// TIA Portal project "SepSimples" (V16)

(* hardware
DEVICE "S71500/ET200MP station_1"  S7-1500 station
   slot 0: "Rail_0"  Rack  6ES7 590-1***0-0AA0
   slot 1: "PLC_1"  CPU 1512C-1 PN  6ES7 512-1CK00-0AB0  V2.8
      slot 3: "CPU display_1"  6ES7591-1AA00-0AA0
      slot 32768: "PROFINET interface_1"  X1
         slot 32769: "Port_1"  X1 P1
         slot 32770: "Port_2"  X1 P2
      slot 34817: "Virtual CP interface port_1"  Virtual CP interface port  Virtual CP interface port
*)

// ===== PLC "PLC_1"  CPU 1512C-1 PN =====

VAR_GLOBAL   // PLC tag table "Default tag table"
   "alwaysFalse" AT %M0.0 : Bool;
END_VAR

VAR_GLOBAL   // PLC tag table "E_N_Controlavel"
   "FIO_S3" AT %M5.3 : Bool;
   "FIO_S2" AT %M5.2 : Bool;
   "FIO_PA" AT %M5.1 : Bool;
   "FIO_PV" AT %M5.0 : Bool;
   "FIO_S4" AT %M5.5 : Bool;
   "FIO_AT_Fwd" AT %M5.6 : Bool;
   "FIOAT_Rev" AT %M5.7 : Bool;
END_VAR

VAR_GLOBAL   // PLC tag table "Saidas"
   "FIO_Atuador" AT %M10.0 : Bool;
   "FIO_Esteira1" AT %M10.1 : Bool;
   "FIO_Esteira2" AT %M10.2 : Bool;
   "FIO_Esteira3" AT %M10.3 : Bool;
   "FIO_Esteira4" AT %M10.4 : Bool;
END_VAR

DATA_BLOCK "Eventos"   // DB1
{ S7_Optimized_Access := 'TRUE' }
VERSION : 0.1
   VAR
      PV_Ev : Bool;
      PA_Ev : Bool;
      S2_On_Ev : Bool;
      S2_Off_Ev : Bool;
      S3_On_Ev : Bool;
      S3_Off_Ev : Bool;
      AT_Off_Ev : Bool;
      S4_Off_Ev : Bool;
      AT_On_Ev : Bool;
      E1_On_Ev : Bool;
      E1_Off_Ev : Bool;
      E2_On_Ev : Bool;
      E2_Off_Ev : Bool;
      E3_On_Ev : Bool;
      E3_Off_Ev : Bool;
   END_VAR
BEGIN
END_DATA_BLOCK

DATA_BLOCK "BitsAuxiliares"   // DB2
{ S7_Optimized_Access := 'TRUE' }
VERSION : 0.1
   VAR
      Aux1 : Bool;
      Aux2 : Bool;
      Aux3 : Bool;
      Aux4 : Bool;
      Aux5 : Bool;
      Aux6 : Bool;
      Aux7 : Bool;
      Aux8 : Bool;
   END_VAR
BEGIN
END_DATA_BLOCK

DATA_BLOCK "EstadosSP"   // DB3
{ S7_Optimized_Access := 'TRUE' }
VERSION : 0.1
   VAR
      GS1_1 : Bool := true;
      GS2_1 : Bool := true;
      GS2_2 : Bool;
      GS3_1 : Bool := true;
      GS3_2 : Bool;
      GAT_1 : Bool := true;
      GAT_2 : Bool;
      GE1_1 : Bool := true;
      GE1_2 : Bool;
      GE2_1 : Bool := true;
      GE2_2 : Bool;
      GE3_1 : Bool := true;
      GE3_2 : Bool;
      GS4_1 : Bool := true;
   END_VAR
BEGIN
END_DATA_BLOCK

DATA_BLOCK "EstadosSup"   // DB4
{ S7_Optimized_Access := 'TRUE' }
VERSION : 0.1
   VAR
      Sup1_1 : Bool := true;
      Sup1_2 : Bool;
      Sup2_1 : Bool := true;
      Sup2_2 : Bool;
      Sup3_1 : Bool := true;
      Sup3_2 : Bool;
      Sup4_1 : Bool := true;
      Sup4_2 : Bool;
      Sup5_1 : Bool := true;
      Sup5_2 : Bool;
      Sup6_1 : Bool := true;
      Sup6_2 : Bool;
      Sup7_1 : Bool := true;
      Sup7_2 : Bool;
      Sup8_1 : Bool := true;
      Sup8_2 : Bool;
      Sup9_1 : Bool := true;
      Sup9_2 : Bool;
      Sup9_3 : Bool;
      Sup10_1 : Bool := true;
      Sup10_2 : Bool;
      Sup10_3 : Bool;
      Sup10_4 : Bool;
   END_VAR
BEGIN
END_DATA_BLOCK

DATA_BLOCK "Des_Eventos"   // DB5
{ S7_Optimized_Access := 'TRUE' }
VERSION : 0.1
   VAR
      d_AT_On : Bool;
      d_E1_On : Bool;
      d_E1_Off : Bool;
      d_E2_On : Bool;
      d_E2_Off : Bool;
      d_E3_On : Bool;
      d_E3_Off : Bool;
   END_VAR
BEGIN
END_DATA_BLOCK

FUNCTION "LeituraEntradas" : Void   // FC2, LAD
TITLE = Leitura das entradas dos eventos não controláveis
{ S7_Optimized_Access := 'TRUE' }
VERSION : 0.1
   VAR_TEMP   // added for the SCL form of the ladder/FBD networks
      _w1 : Bool;
   END_VAR
BEGIN

REGION Network 1: Leitura peça verde
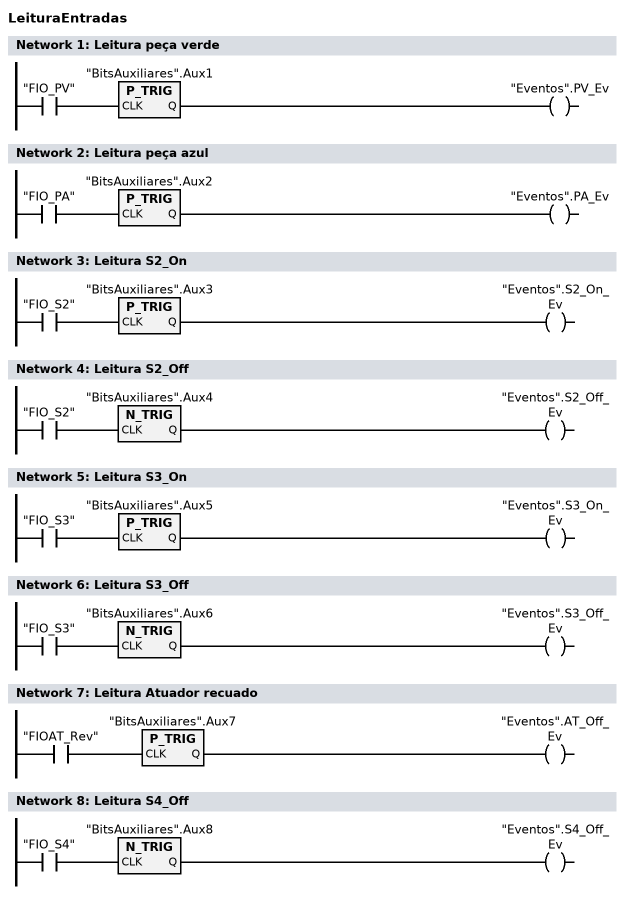
   RUNG wire#powerrail
      Contact( "FIO_PV" )
      P_Trig( "BitsAuxiliares".Aux1 )
      Coil( "Eventos".PV_Ev )
   END_RUNG
   // the same network as SCL:
   #_w1 := "FIO_PV" AND NOT "BitsAuxiliares".Aux1;   // rising edge
   "BitsAuxiliares".Aux1 := "FIO_PV";
   "Eventos".PV_Ev := #_w1;
END_REGION

REGION Network 2: Leitura peça azul
   RUNG wire#powerrail
      Contact( "FIO_PA" )
      P_Trig( "BitsAuxiliares".Aux2 )
      Coil( "Eventos".PA_Ev )
   END_RUNG
   // the same network as SCL:
   #_w1 := "FIO_PA" AND NOT "BitsAuxiliares".Aux2;   // rising edge
   "BitsAuxiliares".Aux2 := "FIO_PA";
   "Eventos".PA_Ev := #_w1;
END_REGION

REGION Network 3: Leitura S2_On
   RUNG wire#powerrail
      Contact( "FIO_S2" )
      P_Trig( "BitsAuxiliares".Aux3 )
      Coil( "Eventos".S2_On_Ev )
   END_RUNG
   // the same network as SCL:
   #_w1 := "FIO_S2" AND NOT "BitsAuxiliares".Aux3;   // rising edge
   "BitsAuxiliares".Aux3 := "FIO_S2";
   "Eventos".S2_On_Ev := #_w1;
END_REGION

REGION Network 4: Leitura S2_Off
   RUNG wire#powerrail
      Contact( "FIO_S2" )
      N_Trig( "BitsAuxiliares".Aux4 )
      Coil( "Eventos".S2_Off_Ev )
   END_RUNG
   // the same network as SCL:
   #_w1 := NOT "FIO_S2" AND "BitsAuxiliares".Aux4;   // falling edge
   "BitsAuxiliares".Aux4 := "FIO_S2";
   "Eventos".S2_Off_Ev := #_w1;
END_REGION

REGION Network 5: Leitura S3_On
   RUNG wire#powerrail
      Contact( "FIO_S3" )
      P_Trig( "BitsAuxiliares".Aux5 )
      Coil( "Eventos".S3_On_Ev )
   END_RUNG
   // the same network as SCL:
   #_w1 := "FIO_S3" AND NOT "BitsAuxiliares".Aux5;   // rising edge
   "BitsAuxiliares".Aux5 := "FIO_S3";
   "Eventos".S3_On_Ev := #_w1;
END_REGION

REGION Network 6: Leitura S3_Off
   RUNG wire#powerrail
      Contact( "FIO_S3" )
      N_Trig( "BitsAuxiliares".Aux6 )
      Coil( "Eventos".S3_Off_Ev )
   END_RUNG
   // the same network as SCL:
   #_w1 := NOT "FIO_S3" AND "BitsAuxiliares".Aux6;   // falling edge
   "BitsAuxiliares".Aux6 := "FIO_S3";
   "Eventos".S3_Off_Ev := #_w1;
END_REGION

REGION Network 7: Leitura Atuador recuado
   RUNG wire#powerrail
      Contact( "FIOAT_Rev" )
      P_Trig( "BitsAuxiliares".Aux7 )
      Coil( "Eventos".AT_Off_Ev )
   END_RUNG
   // the same network as SCL:
   #_w1 := "FIOAT_Rev" AND NOT "BitsAuxiliares".Aux7;   // rising edge
   "BitsAuxiliares".Aux7 := "FIOAT_Rev";
   "Eventos".AT_Off_Ev := #_w1;
END_REGION

REGION Network 8: Leitura S4_Off
   RUNG wire#powerrail
      Contact( "FIO_S4" )
      N_Trig( "BitsAuxiliares".Aux8 )
      Coil( "Eventos".S4_Off_Ev )
   END_RUNG
   // the same network as SCL:
   #_w1 := NOT "FIO_S4" AND "BitsAuxiliares".Aux8;   // falling edge
   "BitsAuxiliares".Aux8 := "FIO_S4";
   "Eventos".S4_Off_Ev := #_w1;
END_REGION
END_FUNCTION

FUNCTION "At_SP_NaoControlaveis" : Void   // FC3, LAD
TITLE = Atualização dos estados do sistema produto a partir dos eventos não controláveis.
{ S7_Optimized_Access := 'TRUE' }
VERSION : 0.1
BEGIN

REGION Network 1: Modelo de S2, do estado 1 para o estado 2.
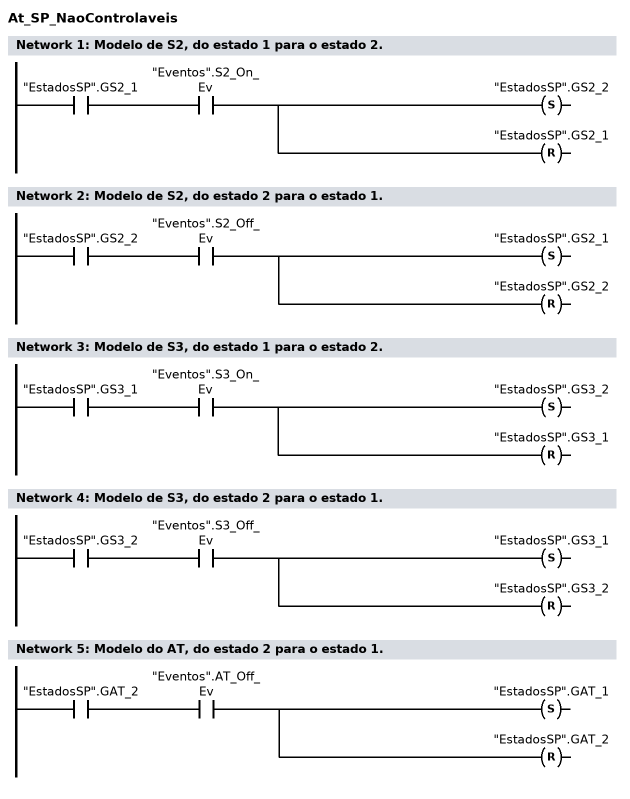
   RUNG wire#powerrail
      Contact( "EstadosSP".GS2_1 )
      Contact( "Eventos".S2_On_Ev )
      wire#w1
      S_Coil( "EstadosSP".GS2_2 )
   END_RUNG
   RUNG wire#w1
      R_Coil( "EstadosSP".GS2_1 )
   END_RUNG
   // the same network as SCL:
   IF "EstadosSP".GS2_1 AND "Eventos".S2_On_Ev THEN
       "EstadosSP".GS2_2 := TRUE;
       "EstadosSP".GS2_1 := FALSE;
   END_IF;
END_REGION

REGION Network 2: Modelo de S2, do estado 2 para o estado 1.
   RUNG wire#powerrail
      Contact( "EstadosSP".GS2_2 )
      Contact( "Eventos".S2_Off_Ev )
      wire#w1
      S_Coil( "EstadosSP".GS2_1 )
   END_RUNG
   RUNG wire#w1
      R_Coil( "EstadosSP".GS2_2 )
   END_RUNG
   // the same network as SCL:
   IF "EstadosSP".GS2_2 AND "Eventos".S2_Off_Ev THEN
       "EstadosSP".GS2_1 := TRUE;
       "EstadosSP".GS2_2 := FALSE;
   END_IF;
END_REGION

REGION Network 3: Modelo de S3, do estado 1 para o estado 2.
   RUNG wire#powerrail
      Contact( "EstadosSP".GS3_1 )
      Contact( "Eventos".S3_On_Ev )
      wire#w1
      S_Coil( "EstadosSP".GS3_2 )
   END_RUNG
   RUNG wire#w1
      R_Coil( "EstadosSP".GS3_1 )
   END_RUNG
   // the same network as SCL:
   IF "EstadosSP".GS3_1 AND "Eventos".S3_On_Ev THEN
       "EstadosSP".GS3_2 := TRUE;
       "EstadosSP".GS3_1 := FALSE;
   END_IF;
END_REGION

REGION Network 4: Modelo de S3, do estado 2 para o estado 1.
   RUNG wire#powerrail
      Contact( "EstadosSP".GS3_2 )
      Contact( "Eventos".S3_Off_Ev )
      wire#w1
      S_Coil( "EstadosSP".GS3_1 )
   END_RUNG
   RUNG wire#w1
      R_Coil( "EstadosSP".GS3_2 )
   END_RUNG
   // the same network as SCL:
   IF "EstadosSP".GS3_2 AND "Eventos".S3_Off_Ev THEN
       "EstadosSP".GS3_1 := TRUE;
       "EstadosSP".GS3_2 := FALSE;
   END_IF;
END_REGION

REGION Network 5: Modelo do AT, do estado 2 para o estado 1.
   RUNG wire#powerrail
      Contact( "EstadosSP".GAT_2 )
      Contact( "Eventos".AT_Off_Ev )
      wire#w1
      S_Coil( "EstadosSP".GAT_1 )
   END_RUNG
   RUNG wire#w1
      R_Coil( "EstadosSP".GAT_2 )
   END_RUNG
   // the same network as SCL:
   IF "EstadosSP".GAT_2 AND "Eventos".AT_Off_Ev THEN
       "EstadosSP".GAT_1 := TRUE;
       "EstadosSP".GAT_2 := FALSE;
   END_IF;
END_REGION
END_FUNCTION

FUNCTION "At_Sup_NaoControlaveis" : Void   // FC4, LAD
TITLE = Atualização dos estados dos supervisores reduzidos, devido a eventos não controláveis
{ S7_Optimized_Access := 'TRUE' }
VERSION : 0.1
BEGIN

REGION Network 1: Atualização do supervisor 1, estado 2 para estado 1.
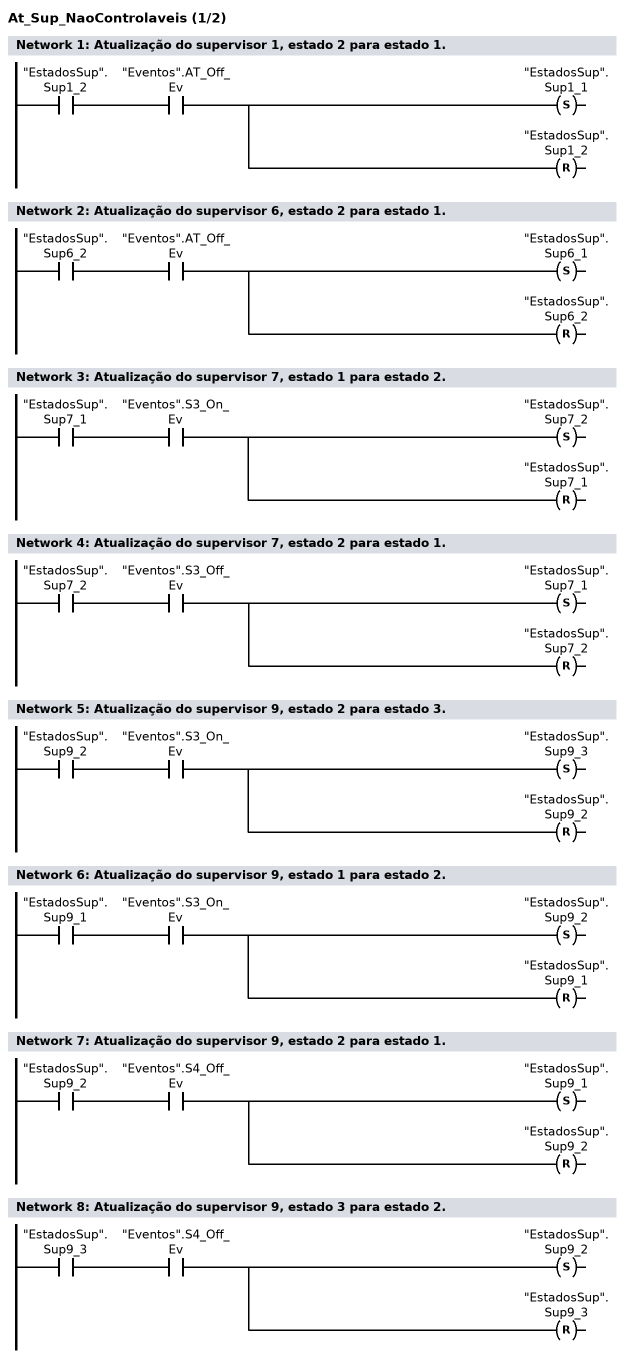
   RUNG wire#powerrail
      Contact( "EstadosSup".Sup1_2 )
      Contact( "Eventos".AT_Off_Ev )
      wire#w1
      S_Coil( "EstadosSup".Sup1_1 )
   END_RUNG
   RUNG wire#w1
      R_Coil( "EstadosSup".Sup1_2 )
   END_RUNG
   // the same network as SCL:
   IF "EstadosSup".Sup1_2 AND "Eventos".AT_Off_Ev THEN
       "EstadosSup".Sup1_1 := TRUE;
       "EstadosSup".Sup1_2 := FALSE;
   END_IF;
END_REGION

REGION Network 2: Atualização do supervisor 6, estado 2 para estado 1.
   RUNG wire#powerrail
      Contact( "EstadosSup".Sup6_2 )
      Contact( "Eventos".AT_Off_Ev )
      wire#w1
      S_Coil( "EstadosSup".Sup6_1 )
   END_RUNG
   RUNG wire#w1
      R_Coil( "EstadosSup".Sup6_2 )
   END_RUNG
   // the same network as SCL:
   IF "EstadosSup".Sup6_2 AND "Eventos".AT_Off_Ev THEN
       "EstadosSup".Sup6_1 := TRUE;
       "EstadosSup".Sup6_2 := FALSE;
   END_IF;
END_REGION

REGION Network 3: Atualização do supervisor 7, estado 1 para estado 2.
   RUNG wire#powerrail
      Contact( "EstadosSup".Sup7_1 )
      Contact( "Eventos".S3_On_Ev )
      wire#w1
      S_Coil( "EstadosSup".Sup7_2 )
   END_RUNG
   RUNG wire#w1
      R_Coil( "EstadosSup".Sup7_1 )
   END_RUNG
   // the same network as SCL:
   IF "EstadosSup".Sup7_1 AND "Eventos".S3_On_Ev THEN
       "EstadosSup".Sup7_2 := TRUE;
       "EstadosSup".Sup7_1 := FALSE;
   END_IF;
END_REGION

REGION Network 4: Atualização do supervisor 7, estado 2 para estado 1.
   RUNG wire#powerrail
      Contact( "EstadosSup".Sup7_2 )
      Contact( "Eventos".S3_Off_Ev )
      wire#w1
      S_Coil( "EstadosSup".Sup7_1 )
   END_RUNG
   RUNG wire#w1
      R_Coil( "EstadosSup".Sup7_2 )
   END_RUNG
   // the same network as SCL:
   IF "EstadosSup".Sup7_2 AND "Eventos".S3_Off_Ev THEN
       "EstadosSup".Sup7_1 := TRUE;
       "EstadosSup".Sup7_2 := FALSE;
   END_IF;
END_REGION

REGION Network 5: Atualização do supervisor 9, estado 2 para estado 3.
   RUNG wire#powerrail
      Contact( "EstadosSup".Sup9_2 )
      Contact( "Eventos".S3_On_Ev )
      wire#w1
      S_Coil( "EstadosSup".Sup9_3 )
   END_RUNG
   RUNG wire#w1
      R_Coil( "EstadosSup".Sup9_2 )
   END_RUNG
   // the same network as SCL:
   IF "EstadosSup".Sup9_2 AND "Eventos".S3_On_Ev THEN
       "EstadosSup".Sup9_3 := TRUE;
       "EstadosSup".Sup9_2 := FALSE;
   END_IF;
END_REGION

REGION Network 6: Atualização do supervisor 9, estado 1 para estado 2.
   RUNG wire#powerrail
      Contact( "EstadosSup".Sup9_1 )
      Contact( "Eventos".S3_On_Ev )
      wire#w1
      S_Coil( "EstadosSup".Sup9_2 )
   END_RUNG
   RUNG wire#w1
      R_Coil( "EstadosSup".Sup9_1 )
   END_RUNG
   // the same network as SCL:
   IF "EstadosSup".Sup9_1 AND "Eventos".S3_On_Ev THEN
       "EstadosSup".Sup9_2 := TRUE;
       "EstadosSup".Sup9_1 := FALSE;
   END_IF;
END_REGION

REGION Network 7: Atualização do supervisor 9, estado 2 para estado 1.
   RUNG wire#powerrail
      Contact( "EstadosSup".Sup9_2 )
      Contact( "Eventos".S4_Off_Ev )
      wire#w1
      S_Coil( "EstadosSup".Sup9_1 )
   END_RUNG
   RUNG wire#w1
      R_Coil( "EstadosSup".Sup9_2 )
   END_RUNG
   // the same network as SCL:
   IF "EstadosSup".Sup9_2 AND "Eventos".S4_Off_Ev THEN
       "EstadosSup".Sup9_1 := TRUE;
       "EstadosSup".Sup9_2 := FALSE;
   END_IF;
END_REGION

REGION Network 8: Atualização do supervisor 9, estado 3 para estado 2.
   RUNG wire#powerrail
      Contact( "EstadosSup".Sup9_3 )
      Contact( "Eventos".S4_Off_Ev )
      wire#w1
      S_Coil( "EstadosSup".Sup9_2 )
   END_RUNG
   RUNG wire#w1
      R_Coil( "EstadosSup".Sup9_3 )
   END_RUNG
   // the same network as SCL:
   IF "EstadosSup".Sup9_3 AND "Eventos".S4_Off_Ev THEN
       "EstadosSup".Sup9_2 := TRUE;
       "EstadosSup".Sup9_3 := FALSE;
   END_IF;
END_REGION

REGION Network 9: Atualização do supervisor 10, estado 1 para estado 2.
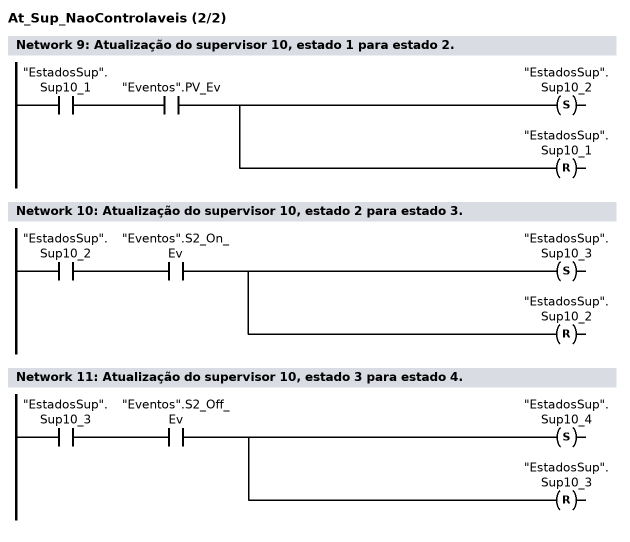
   RUNG wire#powerrail
      Contact( "EstadosSup".Sup10_1 )
      Contact( "Eventos".PV_Ev )
      wire#w1
      S_Coil( "EstadosSup".Sup10_2 )
   END_RUNG
   RUNG wire#w1
      R_Coil( "EstadosSup".Sup10_1 )
   END_RUNG
   // the same network as SCL:
   IF "EstadosSup".Sup10_1 AND "Eventos".PV_Ev THEN
       "EstadosSup".Sup10_2 := TRUE;
       "EstadosSup".Sup10_1 := FALSE;
   END_IF;
END_REGION

REGION Network 10: Atualização do supervisor 10, estado 2 para estado 3.
   RUNG wire#powerrail
      Contact( "EstadosSup".Sup10_2 )
      Contact( "Eventos".S2_On_Ev )
      wire#w1
      S_Coil( "EstadosSup".Sup10_3 )
   END_RUNG
   RUNG wire#w1
      R_Coil( "EstadosSup".Sup10_2 )
   END_RUNG
   // the same network as SCL:
   IF "EstadosSup".Sup10_2 AND "Eventos".S2_On_Ev THEN
       "EstadosSup".Sup10_3 := TRUE;
       "EstadosSup".Sup10_2 := FALSE;
   END_IF;
END_REGION

REGION Network 11: Atualização do supervisor 10, estado 3 para estado 4.
   RUNG wire#powerrail
      Contact( "EstadosSup".Sup10_3 )
      Contact( "Eventos".S2_Off_Ev )
      wire#w1
      S_Coil( "EstadosSup".Sup10_4 )
   END_RUNG
   RUNG wire#w1
      R_Coil( "EstadosSup".Sup10_3 )
   END_RUNG
   // the same network as SCL:
   IF "EstadosSup".Sup10_3 AND "Eventos".S2_Off_Ev THEN
       "EstadosSup".Sup10_4 := TRUE;
       "EstadosSup".Sup10_3 := FALSE;
   END_IF;
END_REGION
END_FUNCTION

FUNCTION "Des_EventosControlaveis" : Void   // FC5, LAD
TITLE = Desativação dos eventos controláveis
{ S7_Optimized_Access := 'TRUE' }
VERSION : 0.1
BEGIN

REGION Network 1: Desabilita o avança atuador
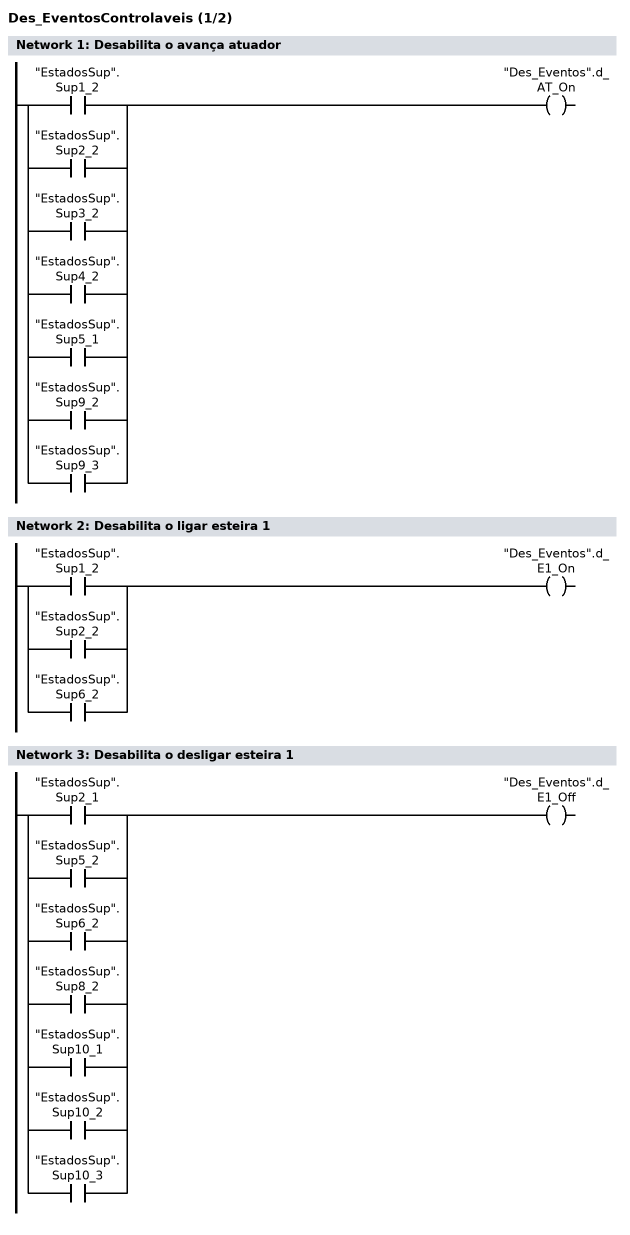
   RUNG wire#powerrail
      Contact( "EstadosSup".Sup1_2 )
      wire#w1
      Coil( "Des_Eventos".d_AT_On )
   END_RUNG
   RUNG wire#powerrail
      Contact( "EstadosSup".Sup2_2 )
   END_RUNG wire#w1
   RUNG wire#powerrail
      Contact( "EstadosSup".Sup3_2 )
   END_RUNG wire#w1
   RUNG wire#powerrail
      Contact( "EstadosSup".Sup4_2 )
   END_RUNG wire#w1
   RUNG wire#powerrail
      Contact( "EstadosSup".Sup5_1 )
   END_RUNG wire#w1
   RUNG wire#powerrail
      Contact( "EstadosSup".Sup9_2 )
   END_RUNG wire#w1
   RUNG wire#powerrail
      Contact( "EstadosSup".Sup9_3 )
   END_RUNG wire#w1
   // the same network as SCL:
   "Des_Eventos".d_AT_On := "EstadosSup".Sup1_2 OR "EstadosSup".Sup2_2 OR "EstadosSup".Sup3_2 OR "EstadosSup".Sup4_2 OR "EstadosSup".Sup5_1 OR "EstadosSup".Sup9_2 OR "EstadosSup".Sup9_3;
END_REGION

REGION Network 2: Desabilita o ligar esteira 1
   RUNG wire#powerrail
      Contact( "EstadosSup".Sup1_2 )
      wire#w1
      Coil( "Des_Eventos".d_E1_On )
   END_RUNG
   RUNG wire#powerrail
      Contact( "EstadosSup".Sup2_2 )
   END_RUNG wire#w1
   RUNG wire#powerrail
      Contact( "EstadosSup".Sup6_2 )
   END_RUNG wire#w1
   // the same network as SCL:
   "Des_Eventos".d_E1_On := "EstadosSup".Sup1_2 OR "EstadosSup".Sup2_2 OR "EstadosSup".Sup6_2;
END_REGION

REGION Network 3: Desabilita o desligar esteira 1
   RUNG wire#powerrail
      Contact( "EstadosSup".Sup2_1 )
      wire#w1
      Coil( "Des_Eventos".d_E1_Off )
   END_RUNG
   RUNG wire#powerrail
      Contact( "EstadosSup".Sup5_2 )
   END_RUNG wire#w1
   RUNG wire#powerrail
      Contact( "EstadosSup".Sup6_2 )
   END_RUNG wire#w1
   RUNG wire#powerrail
      Contact( "EstadosSup".Sup8_2 )
   END_RUNG wire#w1
   RUNG wire#powerrail
      Contact( "EstadosSup".Sup10_1 )
   END_RUNG wire#w1
   RUNG wire#powerrail
      Contact( "EstadosSup".Sup10_2 )
   END_RUNG wire#w1
   RUNG wire#powerrail
      Contact( "EstadosSup".Sup10_3 )
   END_RUNG wire#w1
   // the same network as SCL:
   "Des_Eventos".d_E1_Off := "EstadosSup".Sup2_1 OR "EstadosSup".Sup5_2 OR "EstadosSup".Sup6_2 OR "EstadosSup".Sup8_2 OR "EstadosSup".Sup10_1 OR "EstadosSup".Sup10_2 OR "EstadosSup".Sup10_3;
END_REGION

REGION Network 4: Desabilita o ligar esteira 2
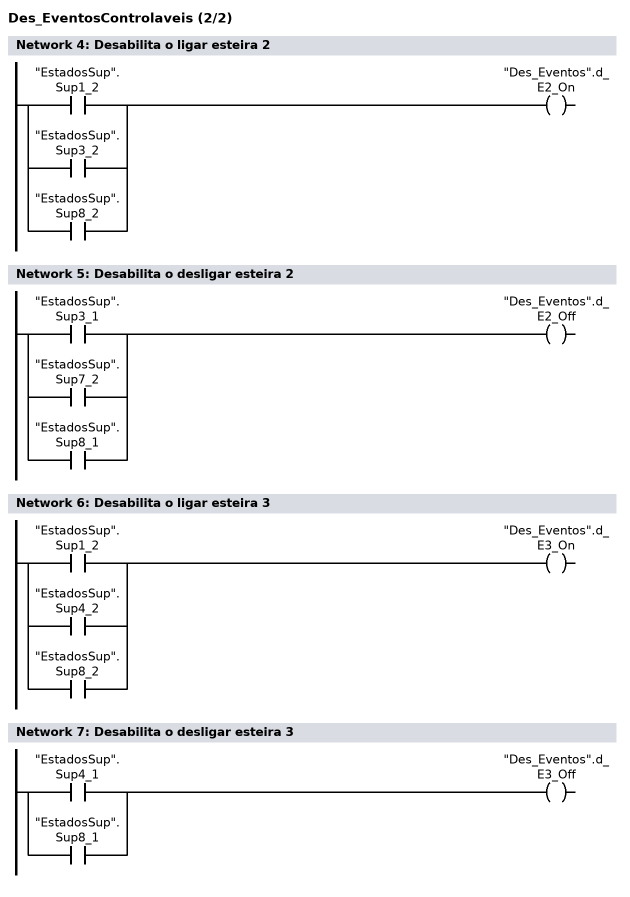
   RUNG wire#powerrail
      Contact( "EstadosSup".Sup1_2 )
      wire#w1
      Coil( "Des_Eventos".d_E2_On )
   END_RUNG
   RUNG wire#powerrail
      Contact( "EstadosSup".Sup3_2 )
   END_RUNG wire#w1
   RUNG wire#powerrail
      Contact( "EstadosSup".Sup8_2 )
   END_RUNG wire#w1
   // the same network as SCL:
   "Des_Eventos".d_E2_On := "EstadosSup".Sup1_2 OR "EstadosSup".Sup3_2 OR "EstadosSup".Sup8_2;
END_REGION

REGION Network 5: Desabilita o desligar esteira 2
   RUNG wire#powerrail
      Contact( "EstadosSup".Sup3_1 )
      wire#w1
      Coil( "Des_Eventos".d_E2_Off )
   END_RUNG
   RUNG wire#powerrail
      Contact( "EstadosSup".Sup7_2 )
   END_RUNG wire#w1
   RUNG wire#powerrail
      Contact( "EstadosSup".Sup8_1 )
   END_RUNG wire#w1
   // the same network as SCL:
   "Des_Eventos".d_E2_Off := "EstadosSup".Sup3_1 OR "EstadosSup".Sup7_2 OR "EstadosSup".Sup8_1;
END_REGION

REGION Network 6: Desabilita o ligar esteira 3
   RUNG wire#powerrail
      Contact( "EstadosSup".Sup1_2 )
      wire#w1
      Coil( "Des_Eventos".d_E3_On )
   END_RUNG
   RUNG wire#powerrail
      Contact( "EstadosSup".Sup4_2 )
   END_RUNG wire#w1
   RUNG wire#powerrail
      Contact( "EstadosSup".Sup8_2 )
   END_RUNG wire#w1
   // the same network as SCL:
   "Des_Eventos".d_E3_On := "EstadosSup".Sup1_2 OR "EstadosSup".Sup4_2 OR "EstadosSup".Sup8_2;
END_REGION

REGION Network 7: Desabilita o desligar esteira 3
   RUNG wire#powerrail
      Contact( "EstadosSup".Sup4_1 )
      wire#w1
      Coil( "Des_Eventos".d_E3_Off )
   END_RUNG
   RUNG wire#powerrail
      Contact( "EstadosSup".Sup8_1 )
   END_RUNG wire#w1
   // the same network as SCL:
   "Des_Eventos".d_E3_Off := "EstadosSup".Sup4_1 OR "EstadosSup".Sup8_1;
END_REGION
END_FUNCTION

FUNCTION "Ger_Eventos_Contr" : Void   // FC6, LAD
TITLE = Geração de eventos controláveis e atualização dos modelos do SP.
{ S7_Optimized_Access := 'TRUE' }
VERSION : 0.1
   VAR_TEMP   // added for the SCL form of the ladder/FBD networks
      _w1 : Bool;
   END_VAR
BEGIN

REGION Network 1: Geração evento de acionar atuador
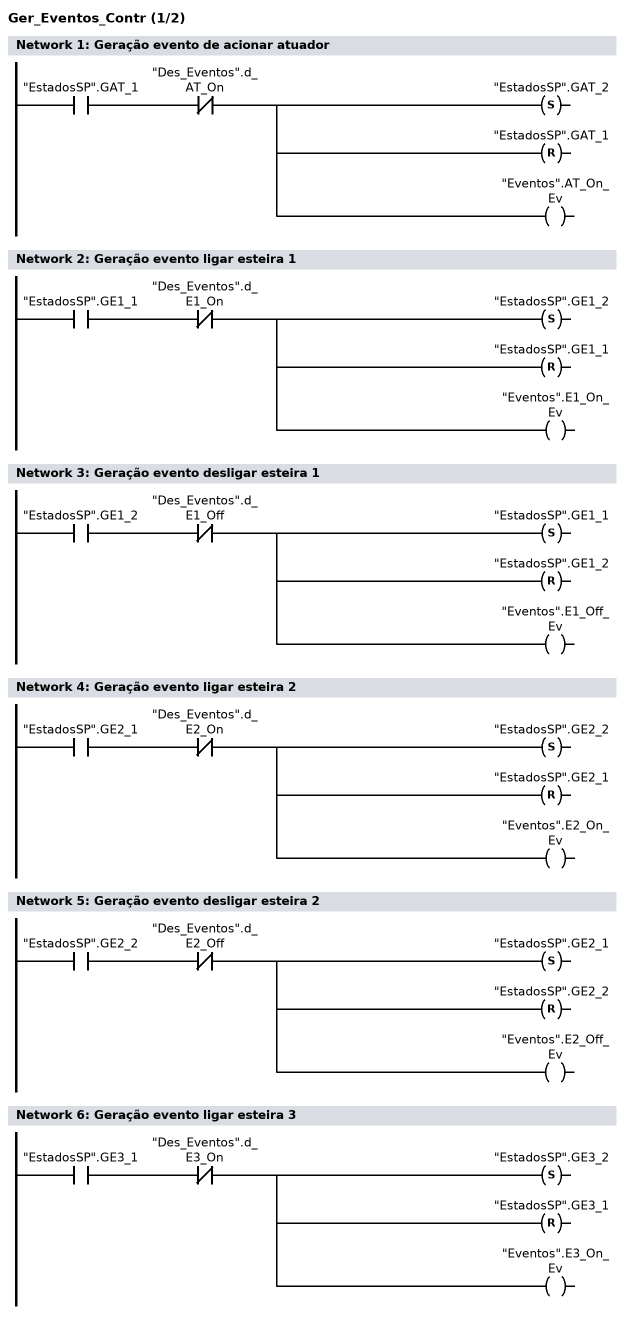
   RUNG wire#powerrail
      Contact( "EstadosSP".GAT_1 )
      I_Contact( "Des_Eventos".d_AT_On )
      wire#w1
      S_Coil( "EstadosSP".GAT_2 )
   END_RUNG
   RUNG wire#w1
      R_Coil( "EstadosSP".GAT_1 )
   END_RUNG
   RUNG wire#w1
      Coil( "Eventos".AT_On_Ev )
   END_RUNG
   // the same network as SCL:
   #_w1 := "EstadosSP".GAT_1 AND NOT "Des_Eventos".d_AT_On;
   IF #_w1 THEN
       "EstadosSP".GAT_2 := TRUE;
       "EstadosSP".GAT_1 := FALSE;
   END_IF;
   "Eventos".AT_On_Ev := #_w1;
END_REGION

REGION Network 2: Geração evento ligar esteira 1
   RUNG wire#powerrail
      Contact( "EstadosSP".GE1_1 )
      I_Contact( "Des_Eventos".d_E1_On )
      wire#w1
      S_Coil( "EstadosSP".GE1_2 )
   END_RUNG
   RUNG wire#w1
      R_Coil( "EstadosSP".GE1_1 )
   END_RUNG
   RUNG wire#w1
      Coil( "Eventos".E1_On_Ev )
   END_RUNG
   // the same network as SCL:
   #_w1 := "EstadosSP".GE1_1 AND NOT "Des_Eventos".d_E1_On;
   IF #_w1 THEN
       "EstadosSP".GE1_2 := TRUE;
       "EstadosSP".GE1_1 := FALSE;
   END_IF;
   "Eventos".E1_On_Ev := #_w1;
END_REGION

REGION Network 3: Geração evento desligar esteira 1
   RUNG wire#powerrail
      Contact( "EstadosSP".GE1_2 )
      I_Contact( "Des_Eventos".d_E1_Off )
      wire#w1
      S_Coil( "EstadosSP".GE1_1 )
   END_RUNG
   RUNG wire#w1
      R_Coil( "EstadosSP".GE1_2 )
   END_RUNG
   RUNG wire#w1
      Coil( "Eventos".E1_Off_Ev )
   END_RUNG
   // the same network as SCL:
   #_w1 := "EstadosSP".GE1_2 AND NOT "Des_Eventos".d_E1_Off;
   IF #_w1 THEN
       "EstadosSP".GE1_1 := TRUE;
       "EstadosSP".GE1_2 := FALSE;
   END_IF;
   "Eventos".E1_Off_Ev := #_w1;
END_REGION

REGION Network 4: Geração evento ligar esteira 2
   RUNG wire#powerrail
      Contact( "EstadosSP".GE2_1 )
      I_Contact( "Des_Eventos".d_E2_On )
      wire#w1
      S_Coil( "EstadosSP".GE2_2 )
   END_RUNG
   RUNG wire#w1
      R_Coil( "EstadosSP".GE2_1 )
   END_RUNG
   RUNG wire#w1
      Coil( "Eventos".E2_On_Ev )
   END_RUNG
   // the same network as SCL:
   #_w1 := "EstadosSP".GE2_1 AND NOT "Des_Eventos".d_E2_On;
   IF #_w1 THEN
       "EstadosSP".GE2_2 := TRUE;
       "EstadosSP".GE2_1 := FALSE;
   END_IF;
   "Eventos".E2_On_Ev := #_w1;
END_REGION

REGION Network 5: Geração evento desligar esteira 2
   RUNG wire#powerrail
      Contact( "EstadosSP".GE2_2 )
      I_Contact( "Des_Eventos".d_E2_Off )
      wire#w1
      S_Coil( "EstadosSP".GE2_1 )
   END_RUNG
   RUNG wire#w1
      R_Coil( "EstadosSP".GE2_2 )
   END_RUNG
   RUNG wire#w1
      Coil( "Eventos".E2_Off_Ev )
   END_RUNG
   // the same network as SCL:
   #_w1 := "EstadosSP".GE2_2 AND NOT "Des_Eventos".d_E2_Off;
   IF #_w1 THEN
       "EstadosSP".GE2_1 := TRUE;
       "EstadosSP".GE2_2 := FALSE;
   END_IF;
   "Eventos".E2_Off_Ev := #_w1;
END_REGION

REGION Network 6: Geração evento ligar esteira 3
   RUNG wire#powerrail
      Contact( "EstadosSP".GE3_1 )
      I_Contact( "Des_Eventos".d_E3_On )
      wire#w1
      S_Coil( "EstadosSP".GE3_2 )
   END_RUNG
   RUNG wire#w1
      R_Coil( "EstadosSP".GE3_1 )
   END_RUNG
   RUNG wire#w1
      Coil( "Eventos".E3_On_Ev )
   END_RUNG
   // the same network as SCL:
   #_w1 := "EstadosSP".GE3_1 AND NOT "Des_Eventos".d_E3_On;
   IF #_w1 THEN
       "EstadosSP".GE3_2 := TRUE;
       "EstadosSP".GE3_1 := FALSE;
   END_IF;
   "Eventos".E3_On_Ev := #_w1;
END_REGION

REGION Network 7: Geração evento desligar esteira 3
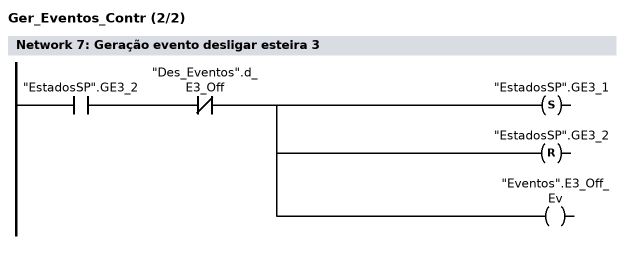
   RUNG wire#powerrail
      Contact( "EstadosSP".GE3_2 )
      I_Contact( "Des_Eventos".d_E3_Off )
      wire#w1
      S_Coil( "EstadosSP".GE3_1 )
   END_RUNG
   RUNG wire#w1
      R_Coil( "EstadosSP".GE3_2 )
   END_RUNG
   RUNG wire#w1
      Coil( "Eventos".E3_Off_Ev )
   END_RUNG
   // the same network as SCL:
   #_w1 := "EstadosSP".GE3_2 AND NOT "Des_Eventos".d_E3_Off;
   IF #_w1 THEN
       "EstadosSP".GE3_1 := TRUE;
       "EstadosSP".GE3_2 := FALSE;
   END_IF;
   "Eventos".E3_Off_Ev := #_w1;
END_REGION
END_FUNCTION

FUNCTION "At_Sup_Controlaveis" : Void   // FC7, LAD
TITLE = Atualização dos estados dos supervisores reduzidos, devido a eventos controláveis
{ S7_Optimized_Access := 'TRUE' }
VERSION : 0.1
   VAR_TEMP   // added for the SCL form of the ladder/FBD networks
      _w1 : Bool;
   END_VAR
BEGIN

REGION Network 1: Atualização do supervisor 1, estado 1 para estado 2.
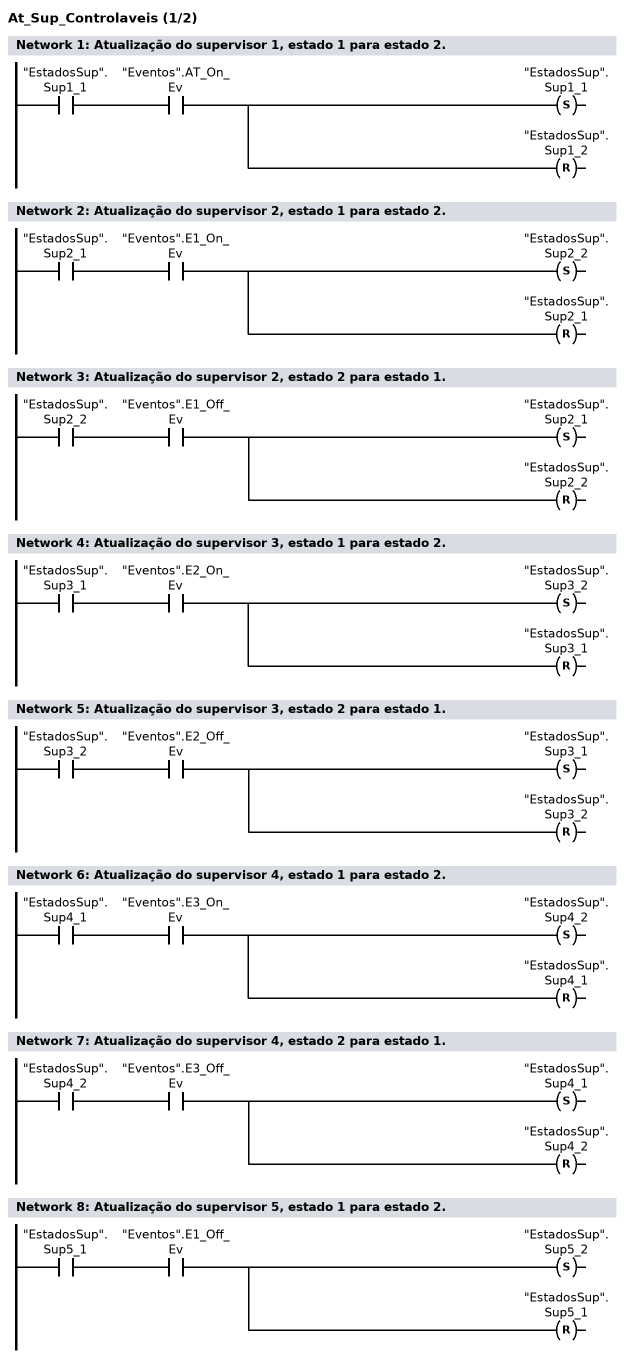
   RUNG wire#powerrail
      Contact( "EstadosSup".Sup1_1 )
      Contact( "Eventos".AT_On_Ev )
      wire#w1
      S_Coil( "EstadosSup".Sup1_1 )
   END_RUNG
   RUNG wire#w1
      R_Coil( "EstadosSup".Sup1_2 )
   END_RUNG
   // the same network as SCL:
   #_w1 := "EstadosSup".Sup1_1 AND "Eventos".AT_On_Ev;
   IF #_w1 THEN
       "EstadosSup".Sup1_1 := TRUE;
       "EstadosSup".Sup1_2 := FALSE;
   END_IF;
END_REGION

REGION Network 2: Atualização do supervisor 2, estado 1 para estado 2.
   RUNG wire#powerrail
      Contact( "EstadosSup".Sup2_1 )
      Contact( "Eventos".E1_On_Ev )
      wire#w1
      S_Coil( "EstadosSup".Sup2_2 )
   END_RUNG
   RUNG wire#w1
      R_Coil( "EstadosSup".Sup2_1 )
   END_RUNG
   // the same network as SCL:
   IF "EstadosSup".Sup2_1 AND "Eventos".E1_On_Ev THEN
       "EstadosSup".Sup2_2 := TRUE;
       "EstadosSup".Sup2_1 := FALSE;
   END_IF;
END_REGION

REGION Network 3: Atualização do supervisor 2, estado 2 para estado 1.
   RUNG wire#powerrail
      Contact( "EstadosSup".Sup2_2 )
      Contact( "Eventos".E1_Off_Ev )
      wire#w1
      S_Coil( "EstadosSup".Sup2_1 )
   END_RUNG
   RUNG wire#w1
      R_Coil( "EstadosSup".Sup2_2 )
   END_RUNG
   // the same network as SCL:
   IF "EstadosSup".Sup2_2 AND "Eventos".E1_Off_Ev THEN
       "EstadosSup".Sup2_1 := TRUE;
       "EstadosSup".Sup2_2 := FALSE;
   END_IF;
END_REGION

REGION Network 4: Atualização do supervisor 3, estado 1 para estado 2.
   RUNG wire#powerrail
      Contact( "EstadosSup".Sup3_1 )
      Contact( "Eventos".E2_On_Ev )
      wire#w1
      S_Coil( "EstadosSup".Sup3_2 )
   END_RUNG
   RUNG wire#w1
      R_Coil( "EstadosSup".Sup3_1 )
   END_RUNG
   // the same network as SCL:
   IF "EstadosSup".Sup3_1 AND "Eventos".E2_On_Ev THEN
       "EstadosSup".Sup3_2 := TRUE;
       "EstadosSup".Sup3_1 := FALSE;
   END_IF;
END_REGION

REGION Network 5: Atualização do supervisor 3, estado 2 para estado 1.
   RUNG wire#powerrail
      Contact( "EstadosSup".Sup3_2 )
      Contact( "Eventos".E2_Off_Ev )
      wire#w1
      S_Coil( "EstadosSup".Sup3_1 )
   END_RUNG
   RUNG wire#w1
      R_Coil( "EstadosSup".Sup3_2 )
   END_RUNG
   // the same network as SCL:
   IF "EstadosSup".Sup3_2 AND "Eventos".E2_Off_Ev THEN
       "EstadosSup".Sup3_1 := TRUE;
       "EstadosSup".Sup3_2 := FALSE;
   END_IF;
END_REGION

REGION Network 6: Atualização do supervisor 4, estado 1 para estado 2.
   RUNG wire#powerrail
      Contact( "EstadosSup".Sup4_1 )
      Contact( "Eventos".E3_On_Ev )
      wire#w1
      S_Coil( "EstadosSup".Sup4_2 )
   END_RUNG
   RUNG wire#w1
      R_Coil( "EstadosSup".Sup4_1 )
   END_RUNG
   // the same network as SCL:
   IF "EstadosSup".Sup4_1 AND "Eventos".E3_On_Ev THEN
       "EstadosSup".Sup4_2 := TRUE;
       "EstadosSup".Sup4_1 := FALSE;
   END_IF;
END_REGION

REGION Network 7: Atualização do supervisor 4, estado 2 para estado 1.
   RUNG wire#powerrail
      Contact( "EstadosSup".Sup4_2 )
      Contact( "Eventos".E3_Off_Ev )
      wire#w1
      S_Coil( "EstadosSup".Sup4_1 )
   END_RUNG
   RUNG wire#w1
      R_Coil( "EstadosSup".Sup4_2 )
   END_RUNG
   // the same network as SCL:
   IF "EstadosSup".Sup4_2 AND "Eventos".E3_Off_Ev THEN
       "EstadosSup".Sup4_1 := TRUE;
       "EstadosSup".Sup4_2 := FALSE;
   END_IF;
END_REGION

REGION Network 8: Atualização do supervisor 5, estado 1 para estado 2.
   RUNG wire#powerrail
      Contact( "EstadosSup".Sup5_1 )
      Contact( "Eventos".E1_Off_Ev )
      wire#w1
      S_Coil( "EstadosSup".Sup5_2 )
   END_RUNG
   RUNG wire#w1
      R_Coil( "EstadosSup".Sup5_1 )
   END_RUNG
   // the same network as SCL:
   IF "EstadosSup".Sup5_1 AND "Eventos".E1_Off_Ev THEN
       "EstadosSup".Sup5_2 := TRUE;
       "EstadosSup".Sup5_1 := FALSE;
   END_IF;
END_REGION

REGION Network 9: Atualização do supervisor 5, estado 2 para estado 1.
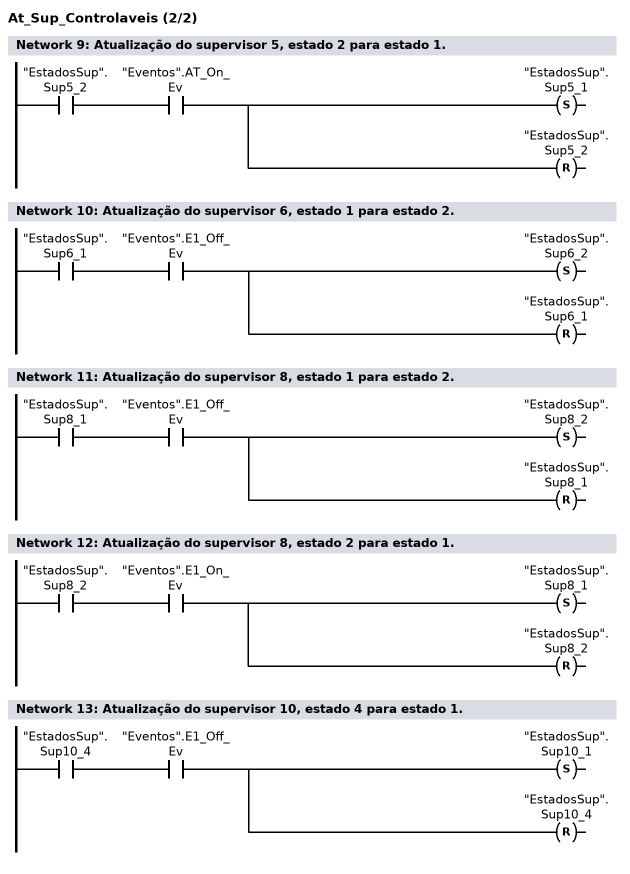
   RUNG wire#powerrail
      Contact( "EstadosSup".Sup5_2 )
      Contact( "Eventos".AT_On_Ev )
      wire#w1
      S_Coil( "EstadosSup".Sup5_1 )
   END_RUNG
   RUNG wire#w1
      R_Coil( "EstadosSup".Sup5_2 )
   END_RUNG
   // the same network as SCL:
   IF "EstadosSup".Sup5_2 AND "Eventos".AT_On_Ev THEN
       "EstadosSup".Sup5_1 := TRUE;
       "EstadosSup".Sup5_2 := FALSE;
   END_IF;
END_REGION

REGION Network 10: Atualização do supervisor 6, estado 1 para estado 2.
   RUNG wire#powerrail
      Contact( "EstadosSup".Sup6_1 )
      Contact( "Eventos".E1_Off_Ev )
      wire#w1
      S_Coil( "EstadosSup".Sup6_2 )
   END_RUNG
   RUNG wire#w1
      R_Coil( "EstadosSup".Sup6_1 )
   END_RUNG
   // the same network as SCL:
   IF "EstadosSup".Sup6_1 AND "Eventos".E1_Off_Ev THEN
       "EstadosSup".Sup6_2 := TRUE;
       "EstadosSup".Sup6_1 := FALSE;
   END_IF;
END_REGION

REGION Network 11: Atualização do supervisor 8, estado 1 para estado 2.
   RUNG wire#powerrail
      Contact( "EstadosSup".Sup8_1 )
      Contact( "Eventos".E1_Off_Ev )
      wire#w1
      S_Coil( "EstadosSup".Sup8_2 )
   END_RUNG
   RUNG wire#w1
      R_Coil( "EstadosSup".Sup8_1 )
   END_RUNG
   // the same network as SCL:
   IF "EstadosSup".Sup8_1 AND "Eventos".E1_Off_Ev THEN
       "EstadosSup".Sup8_2 := TRUE;
       "EstadosSup".Sup8_1 := FALSE;
   END_IF;
END_REGION

REGION Network 12: Atualização do supervisor 8, estado 2 para estado 1.
   RUNG wire#powerrail
      Contact( "EstadosSup".Sup8_2 )
      Contact( "Eventos".E1_On_Ev )
      wire#w1
      S_Coil( "EstadosSup".Sup8_1 )
   END_RUNG
   RUNG wire#w1
      R_Coil( "EstadosSup".Sup8_2 )
   END_RUNG
   // the same network as SCL:
   IF "EstadosSup".Sup8_2 AND "Eventos".E1_On_Ev THEN
       "EstadosSup".Sup8_1 := TRUE;
       "EstadosSup".Sup8_2 := FALSE;
   END_IF;
END_REGION

REGION Network 13: Atualização do supervisor 10, estado 4 para estado 1.
   RUNG wire#powerrail
      Contact( "EstadosSup".Sup10_4 )
      Contact( "Eventos".E1_Off_Ev )
      wire#w1
      S_Coil( "EstadosSup".Sup10_1 )
   END_RUNG
   RUNG wire#w1
      R_Coil( "EstadosSup".Sup10_4 )
   END_RUNG
   // the same network as SCL:
   IF "EstadosSup".Sup10_4 AND "Eventos".E1_Off_Ev THEN
       "EstadosSup".Sup10_1 := TRUE;
       "EstadosSup".Sup10_4 := FALSE;
   END_IF;
END_REGION
END_FUNCTION

FUNCTION "EscritaSaidas" : Void   // FC8, LAD
TITLE = Escrita nos bits de saída
{ S7_Optimized_Access := 'TRUE' }
VERSION : 0.1
BEGIN

REGION Network 1: Atuador
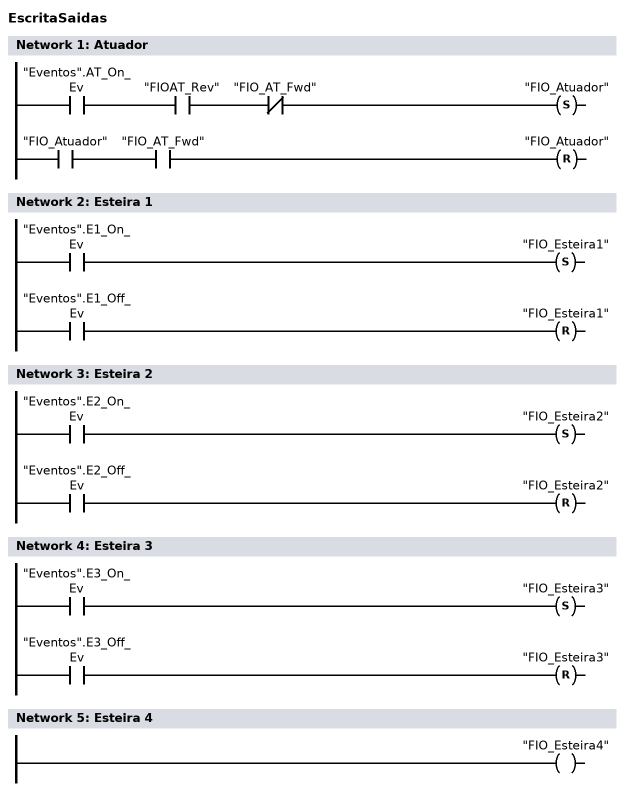
   RUNG wire#powerrail
      Contact( "Eventos".AT_On_Ev )
      Contact( "FIOAT_Rev" )
      I_Contact( "FIO_AT_Fwd" )
      S_Coil( "FIO_Atuador" )
   END_RUNG
   RUNG wire#powerrail
      Contact( "FIO_Atuador" )
      Contact( "FIO_AT_Fwd" )
      R_Coil( "FIO_Atuador" )
   END_RUNG
   // the same network as SCL:
   IF "Eventos".AT_On_Ev AND "FIOAT_Rev" AND NOT "FIO_AT_Fwd" THEN "FIO_Atuador" := TRUE; END_IF;
   IF "FIO_Atuador" AND "FIO_AT_Fwd" THEN "FIO_Atuador" := FALSE; END_IF;
END_REGION

REGION Network 2: Esteira 1
   RUNG wire#powerrail
      Contact( "Eventos".E1_On_Ev )
      S_Coil( "FIO_Esteira1" )
   END_RUNG
   RUNG wire#powerrail
      Contact( "Eventos".E1_Off_Ev )
      R_Coil( "FIO_Esteira1" )
   END_RUNG
   // the same network as SCL:
   IF "Eventos".E1_On_Ev THEN "FIO_Esteira1" := TRUE; END_IF;
   IF "Eventos".E1_Off_Ev THEN "FIO_Esteira1" := FALSE; END_IF;
END_REGION

REGION Network 3: Esteira 2
   RUNG wire#powerrail
      Contact( "Eventos".E2_On_Ev )
      S_Coil( "FIO_Esteira2" )
   END_RUNG
   RUNG wire#powerrail
      Contact( "Eventos".E2_Off_Ev )
      R_Coil( "FIO_Esteira2" )
   END_RUNG
   // the same network as SCL:
   IF "Eventos".E2_On_Ev THEN "FIO_Esteira2" := TRUE; END_IF;
   IF "Eventos".E2_Off_Ev THEN "FIO_Esteira2" := FALSE; END_IF;
END_REGION

REGION Network 4: Esteira 3
   RUNG wire#powerrail
      Contact( "Eventos".E3_On_Ev )
      S_Coil( "FIO_Esteira3" )
   END_RUNG
   RUNG wire#powerrail
      Contact( "Eventos".E3_Off_Ev )
      R_Coil( "FIO_Esteira3" )
   END_RUNG
   // the same network as SCL:
   IF "Eventos".E3_On_Ev THEN "FIO_Esteira3" := TRUE; END_IF;
   IF "Eventos".E3_Off_Ev THEN "FIO_Esteira3" := FALSE; END_IF;
END_REGION

REGION Network 5: Esteira 4
   RUNG wire#powerrail
      Coil( "FIO_Esteira4" )
   END_RUNG
   // the same network as SCL:
   "FIO_Esteira4" := TRUE;
END_REGION
END_FUNCTION

ORGANIZATION_BLOCK "Main"   // OB1, LAD, ProgramCycle
TITLE = "Main Program Sweep (Cycle)"
{ S7_Optimized_Access := 'TRUE' }
VERSION : 0.1
   VAR_INPUT
      Initial_Call : Bool;   // Initial call of this OB
      Remanence : Bool;   // =True, if remanent data are available
   END_VAR
BEGIN

REGION Network 1
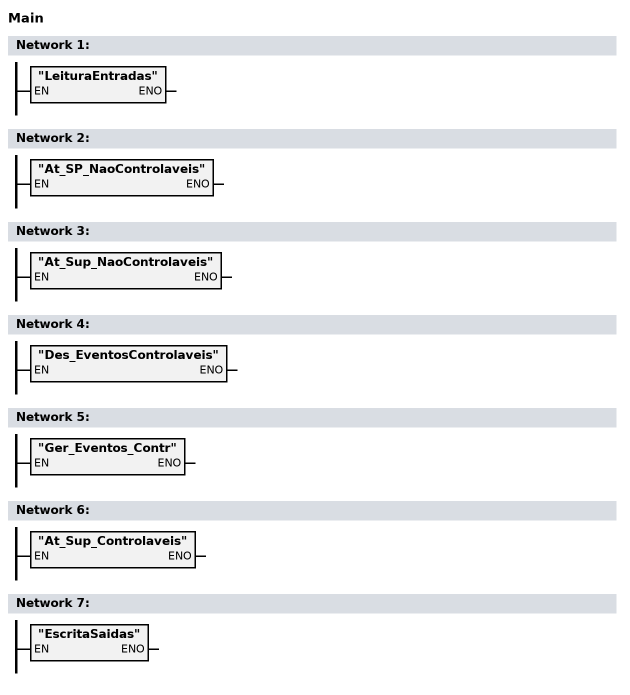
   RUNG wire#powerrail
      "LeituraEntradas"()
   END_RUNG
   // the same network as SCL:
   "LeituraEntradas"();
END_REGION

REGION Network 2
   RUNG wire#powerrail
      "At_SP_NaoControlaveis"()
   END_RUNG
   // the same network as SCL:
   "At_SP_NaoControlaveis"();
END_REGION

REGION Network 3
   RUNG wire#powerrail
      "At_Sup_NaoControlaveis"()
   END_RUNG
   // the same network as SCL:
   "At_Sup_NaoControlaveis"();
END_REGION

REGION Network 4
   RUNG wire#powerrail
      "Des_EventosControlaveis"()
   END_RUNG
   // the same network as SCL:
   "Des_EventosControlaveis"();
END_REGION

REGION Network 5
   RUNG wire#powerrail
      "Ger_Eventos_Contr"()
   END_RUNG
   // the same network as SCL:
   "Ger_Eventos_Contr"();
END_REGION

REGION Network 6
   RUNG wire#powerrail
      "At_Sup_Controlaveis"()
   END_RUNG
   // the same network as SCL:
   "At_Sup_Controlaveis"();
END_REGION

REGION Network 7
   RUNG wire#powerrail
      "EscritaSaidas"()
   END_RUNG
   // the same network as SCL:
   "EscritaSaidas"();
END_REGION
END_ORGANIZATION_BLOCK